(* Schneider Machine Expert - Basic project meccanismo_scelta_spegnimento_graduale_o_livello_minimo, file version 3.0.0.0 *)
(* ProjectInformations: Name=New project *)

HARDWARE
  Cpu 0: TM221C40R
  ModuleExtensionObject 0: TM3AI8/G
  EthernetConfiguration: NetworkName=M221, IpAllocationMode=FixedAddress, IpAddress=0.0.0.0, SubnetMask=0.0.0.0
  SerialLineConfiguration: Baud=Baud19200, Parity=ParityEven, DataBits=DataBits8, StopBits=StopBits1, PhysicalMedium=PhysicalMediumRs485, TransmissionMode=TransmissionModeModbusRtu, SlaveId=1, Addressing=SlaveAddressing
  MastTask: UsePeriodScanMode=false, PeriodScan=100
  FastTask: Period=255
  CpuBehavior: StartingMode=StartAsPreviousState, AutoSaveRamOnEeprom=true, WatchdogPeriod=250

SYMBOLS  (address, symbol, comment, settings)
  %M0       P1_USABILE
  %M1       P2_USABILE
  %M2       P1_COMANDATA  "Stesso valore di P1_CMD. Permette di identificare gli edges, visto che P1_CMD non può farlo."
  %M3       P2_COMANDATA  "Stesso valore di P2_CMD. Permette di identificare gli edges, visto che P2_CMD non può farlo."
  %M4       P3_USABILE
  %M5       P4_USABILE
  %M6       P3_COMANDATA
  %M7       P4_COMANDATA
  %M8       ESISTE_PROX_POMPA_CON_MINOR_ORE  "Nel loop, può non esistere una prossima pompa usabile e non comandata con il minor numero ore."
  %M9       ORA_E_00  "E' mezzanotte?"
  %M10      DECISO_ORDINE  "In intervallo in cui alternare le pompe per altern. giorn., è stata deciso quale sarà prossima pompa con minor ore?"
  %M11      PRIMA_POMPA_COMANDATA  "La prima pompa dell'ordine è stata effettivamente comandata quando serviva?"
  %M12      SECONDA_POMPA_COMANDATA  "La seconda pompa dell'ordine è stata effettivamente comandata quando serviva?"
  %M13      TERZA_POMPA_COMANDATA  "La terza pompa dell'ordine è stata effettivamente comandata quando serviva?"
  %M14      SOTTO_SOGLIA_MIN1
  %M15      SOPRA_SOGLIA_MAX1
  %M16      SOPRA_SOGLIA_MAX2
  %M17      PASSATO_SOGLIA_MAX1
  %M18      PASSATO_SOGLIA_MAX2
  %M19      SOTTO_SOGLIA_MIN2
  %M20      PASSATO_SOGLIA_MAX3
  %M21      PASSATO_SOGLIA_MIN3
  %M22      SOTTO_SOGLIA_MIN3
  %M23      SOPRA_SOGLIA_MAX3
  %M24      P5_USABILE
  %M25        "(occupato, placeholder)"
  %M26      P6_USABILE
  %M27      P5_COMANDATA
  %M28      P6_COMANDATA
  %M29      QUARTA_POMPA_COMANDATA
  %M30      QUINTA_POMPA_COMANDATA
  %M100       "(occupato, placeholder)"
  %MW0      NUM_POMPE_DA_COMANDARE  "Numero di pompe da comandare in base alle soglie raggiunte."
  %MW1      NUM_POMPE_COMANDATE  "Numero di pompe effettivamente comandate, in base alle loro disponibilità."
  %MW2      NUM_POMPE  "Numero di pompe totali."
  %MW3      ULTIMO_MINOR_SECONDI_LAVORATI  "Ultimi secondi lavorati più piccoli (valore temporaneo, da usare solo nel loop)."
  %MW4      PROSSIMA_POMPA_DA_COMANDARE  "Numero da 1 a NUM_POMPE che indica la prossima pompa da comandare."
  %MW5      POMPA_ATTUALE_LOOP  "Pompa attuale nel loop."
  %MW6      NUM_POMPE_COMANDATE_MAX  "Num"
  %MW7      CONTA_POMPE_COMANDATE_MAX  "Da usare in loop e da resettare.  Assume il valore da 1 fino a NUM_POMPE_COMANDATE_MAX."
  %MW8      ORDINE_PRIMA_POMPA
  %MW9      ORDINE_SECONDA_POMPA
  %MW10     ORDINE_TERZA_POMPA
  %MW11     STRG_ALTERNANZA_ATTUALE
  %MW12     LVL_PERC
  %MW13     ORDINE_QUARTA_POMPA
  %MW14     ORDINE_QUINTA_POMPA
  %C0       CONTATORE_P1_SECONDI_LAVORATI  [Preset=0]
  %C1       CONTATORE_P2_SECONDI_LAVORATI  [Preset=0]
  %C2       CONTATORE_P3_SECONDI_LAVORATI  [Preset=0]
  %C3       CONTATORE_P4_SECONDI_LAVORATI  [Preset=0]
  %C4       CONTATORE_P5_SECONDI_LAVORATI  [Preset=0]
  %C5       CONTATORE_P6_SECONDI_LAVORATI  [Preset=0]
  %I0.0     P1_AUTO
  %I0.1     P1_MOTO
  %I0.2     P1_ANOMALIA
  %I0.3     P2_AUTO
  %I0.4     P2_MOTO
  %I0.5     P2_ANOMALIA
  %I0.9     P3_AUTO
  %I0.10    P3_MOTO
  %I0.11    P3_ANOMALIA
  %I0.12    P4_AUTO
  %I0.13    P4_MOTO
  %I0.14    P4_ANOMALIA
  %I0.15    P5_AUTO
  %I0.16    P5_MOTO
  %I0.17    P5_ANOMALIA
  %I0.18    P6_AUTO
  %I0.19    P6_MOTO
  %I0.20    P6_ANOMALIA
  %Q0.0     P1_CMD
  %Q0.1     P2_CMD
  %Q0.2     P3_CMD
  %Q0.3     P4_CMD
  %Q0.4     ERR_STRG_ALTERNANZA_INVALIDA
  %Q0.5     P5_CMD
  %Q0.6     P6_CMD
  %IW0.0    IO_STRG_ALTERNANZA  "0 = livello minimo; 1 = spegnimento graduale;"  [Type=Type_0_10V, Scope=Scope_Normal, Minimum=0, Maximum=1000]
  %IW1.0    IO_LVL  [Type=Type_4_20mA, Scope=Scope_Customized, Minimum=4000, Maximum=20000]
  %IW1.1    SOGLIA_MIN1_PERC  [Type=Type_0_10V, Scope=Scope_Customized, Minimum=0, Maximum=100]
  %IW1.2    SOGLIA_MAX1_PERC  [Type=Type_0_10V, Scope=Scope_Customized, Minimum=0, Maximum=100]
  %IW1.3    SOGLIA_MIN2_PERC  [Type=Type_0_10V, Scope=Scope_Customized, Minimum=0, Maximum=100]
  %IW1.4    SOGLIA_MAX2_PERC  [Type=Type_0_10V, Scope=Scope_Customized, Minimum=0, Maximum=100]
  %IW1.5    SOGLIA_MIN3_PERC  [Type=Type_0_10V, Scope=Scope_Customized, Minimum=0, Maximum=100]
  %IW1.6    SOGLIA_MAX3_PERC  [Type=Type_0_10V, Scope=Scope_Customized, Minimum=0, Maximum=100]

POU Main
  (* SectionNumber=1 *)

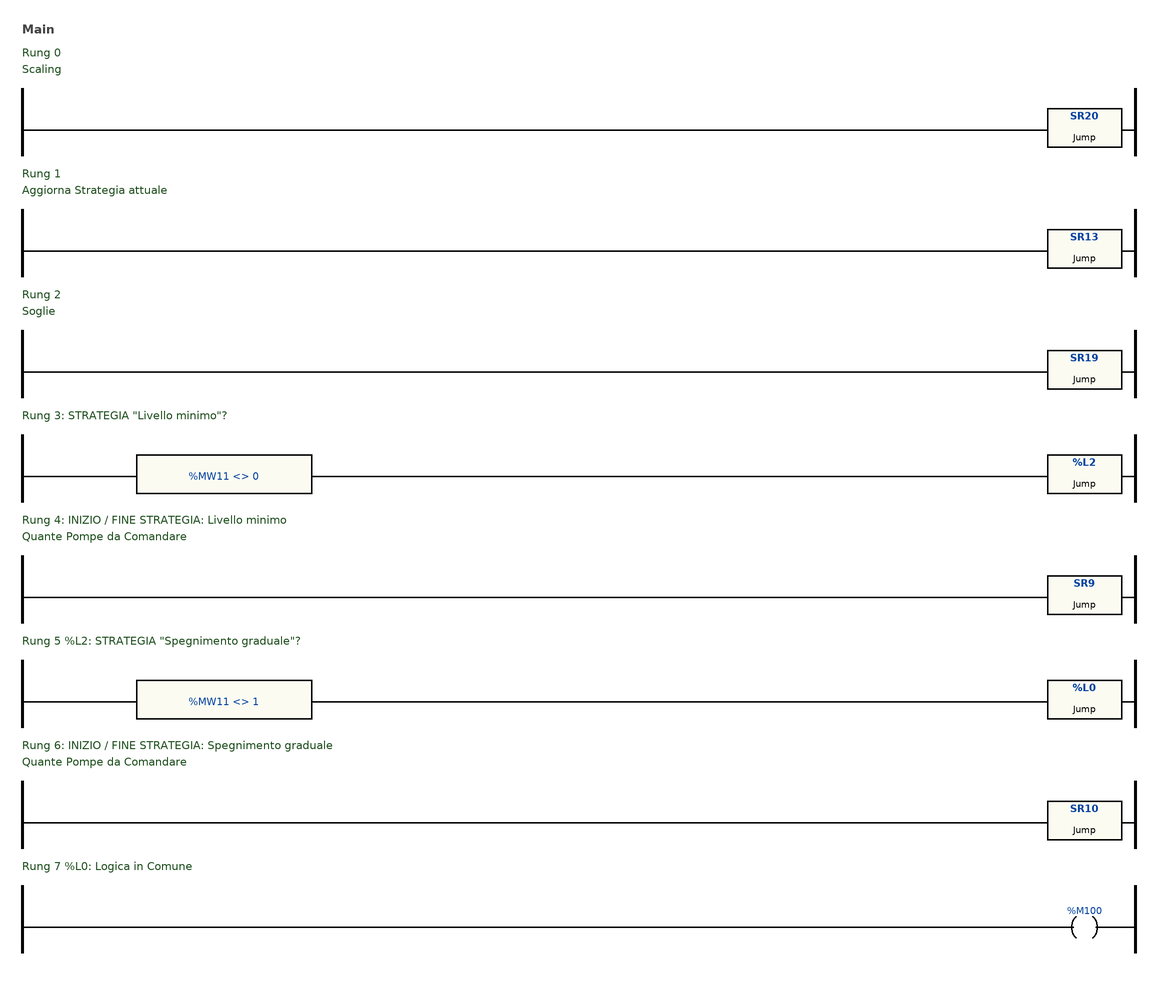

// Rung 0
// Scaling
  LD 1
  SR20
  // as ST:
  //   SR20();

// Rung 1
// Aggiorna Strategia attuale
  LD 1
  SR13
  // as ST:
  //   SR13();

// Rung 2
// Soglie
  LD 1
  SR19
  // as ST:
  //   SR19();

// Rung 3: STRATEGIA "Livello minimo"?
  LD [ %MW11 <> 0 ]       (* STRG_ALTERNANZA_ATTUALE *)
  JMPC %L2
  // as ST:
  //   IF STRG_ALTERNANZA_ATTUALE <> 0 THEN JMP %L2; END_IF;

// Rung 4: INIZIO / FINE STRATEGIA: Livello minimo
// Quante Pompe da Comandare
  LD 1
  SR9
  // as ST:
  //   SR9();

// Rung 5 %L2: STRATEGIA "Spegnimento graduale"?
  %L2:
  LD [ %MW11 <> 1 ]       (* STRG_ALTERNANZA_ATTUALE *)
  JMPC %L0
  // as ST:
  //   %L2:
  //   IF STRG_ALTERNANZA_ATTUALE <> 1 THEN JMP %L0; END_IF;

// Rung 6: INIZIO / FINE STRATEGIA: Spegnimento graduale
// Quante Pompe da Comandare
  LD 1
  SR10
  // as ST:
  //   SR10();

// Rung 7 %L0: Logica in Comune
  %L0:
  LD 1
  ST %M100
  // as ST:
  //   %L0:
  //   %M100 := TRUE;

Subroutine Aggiorna Strategia Alternanza
  (* SectionNumber=11, Number=13 *)

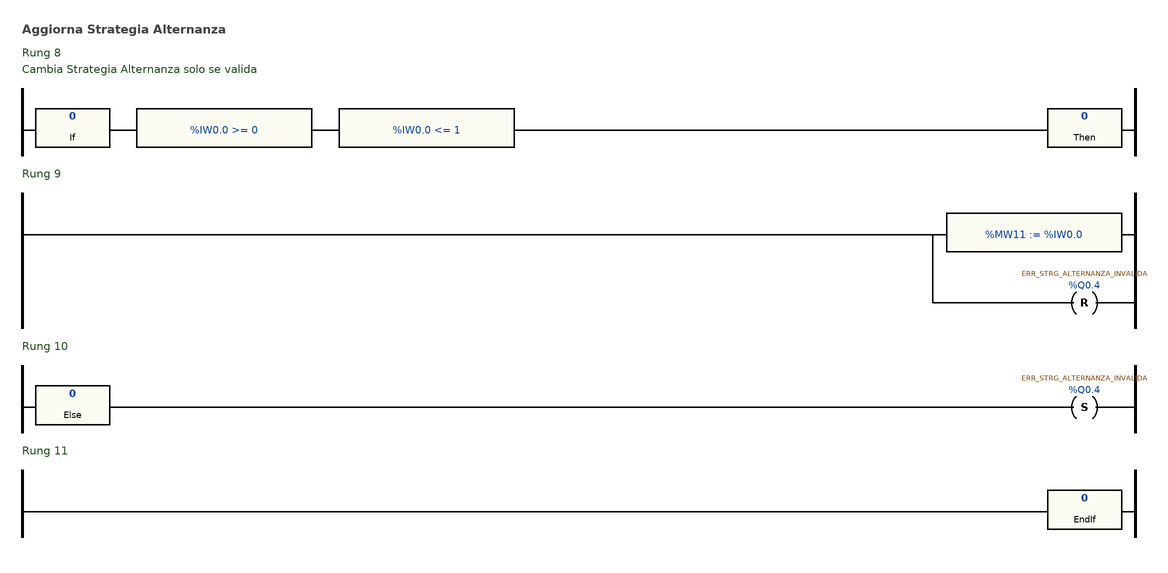

// Rung 8
// Cambia Strategia Alternanza solo se valida
  IF0
  AND [ %IW0.0 >= 0 ]     (* IO_STRG_ALTERNANZA *)
  AND [ %IW0.0 <= 1 ]     (* IO_STRG_ALTERNANZA *)
  THEN0

// Rung 9
  LD 1
  [ %MW11 := %IW0.0 ]     (* STRG_ALTERNANZA_ATTUALE, IO_STRG_ALTERNANZA *)
  R %Q0.4                 (* ERR_STRG_ALTERNANZA_INVALIDA *)
  // as ST:
  //   STRG_ALTERNANZA_ATTUALE := IO_STRG_ALTERNANZA;
  //   ERR_STRG_ALTERNANZA_INVALIDA := FALSE;

// Rung 10
  ELSE0
  S %Q0.4                 (* ERR_STRG_ALTERNANZA_INVALIDA *)

// Rung 11
  LD 1
  ENDIF0

Subroutine Soglie
  (* SectionNumber=12, Number=19 *)

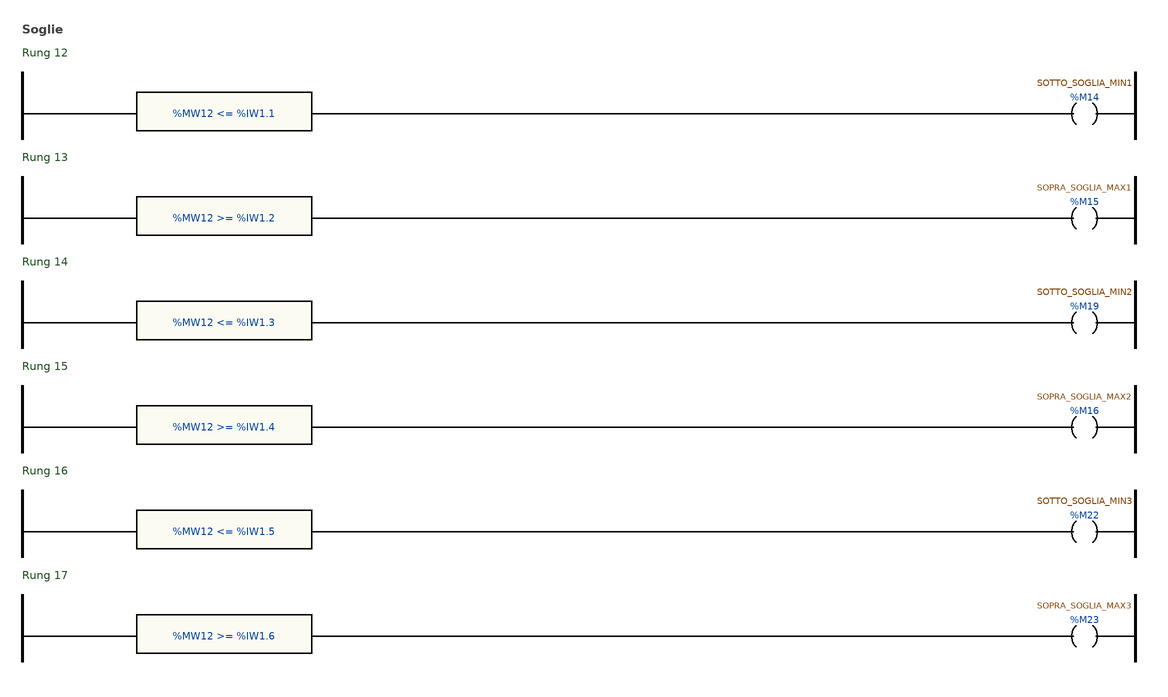

// Rung 12
  LD [ %MW12 <= %IW1.1 ]  (* LVL_PERC, SOGLIA_MIN1_PERC *)
  ST %M14                 (* SOTTO_SOGLIA_MIN1 *)
  // as ST:
  //   SOTTO_SOGLIA_MIN1 := LVL_PERC <= SOGLIA_MIN1_PERC;

// Rung 13
  LD [ %MW12 >= %IW1.2 ]  (* LVL_PERC, SOGLIA_MAX1_PERC *)
  ST %M15                 (* SOPRA_SOGLIA_MAX1 *)
  // as ST:
  //   SOPRA_SOGLIA_MAX1 := LVL_PERC >= SOGLIA_MAX1_PERC;

// Rung 14
  LD [ %MW12 <= %IW1.3 ]  (* LVL_PERC, SOGLIA_MIN2_PERC *)
  ST %M19                 (* SOTTO_SOGLIA_MIN2 *)
  // as ST:
  //   SOTTO_SOGLIA_MIN2 := LVL_PERC <= SOGLIA_MIN2_PERC;

// Rung 15
  LD [ %MW12 >= %IW1.4 ]  (* LVL_PERC, SOGLIA_MAX2_PERC *)
  ST %M16                 (* SOPRA_SOGLIA_MAX2 *)
  // as ST:
  //   SOPRA_SOGLIA_MAX2 := LVL_PERC >= SOGLIA_MAX2_PERC;

// Rung 16
  LD [ %MW12 <= %IW1.5 ]  (* LVL_PERC, SOGLIA_MIN3_PERC *)
  ST %M22                 (* SOTTO_SOGLIA_MIN3 *)
  // as ST:
  //   SOTTO_SOGLIA_MIN3 := LVL_PERC <= SOGLIA_MIN3_PERC;

// Rung 17
  LD [ %MW12 >= %IW1.6 ]  (* LVL_PERC, SOGLIA_MAX3_PERC *)
  ST %M23                 (* SOPRA_SOGLIA_MAX3 *)
  // as ST:
  //   SOPRA_SOGLIA_MAX3 := LVL_PERC >= SOGLIA_MAX3_PERC;

Subroutine Scaling
  (* SectionNumber=13, Number=20 *)

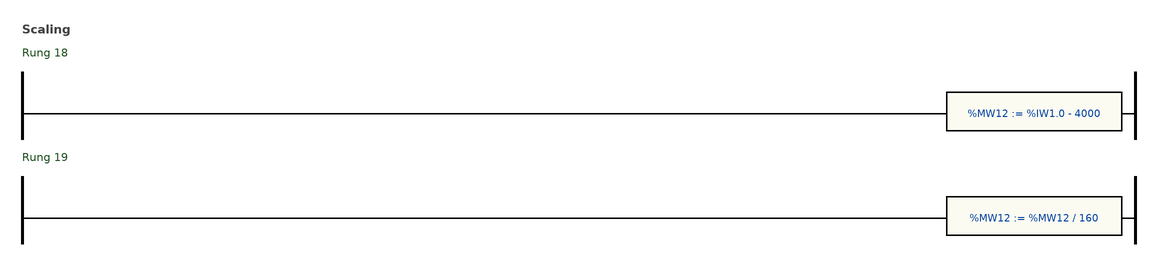

// Rung 18
  LD 1
  [ %MW12 := %IW1.0 - 4000 ](* LVL_PERC, IO_LVL *)
  // as ST:
  //   LVL_PERC := IO_LVL - 4000;

// Rung 19
  LD 1
  [ %MW12 := %MW12 / 160 ](* LVL_PERC, LVL_PERC *)
  // as ST:
  //   LVL_PERC := LVL_PERC / 160;

Subroutine Quante Pompe da Comandare (Livello minimo)
  (* SectionNumber=14, Number=9 *)

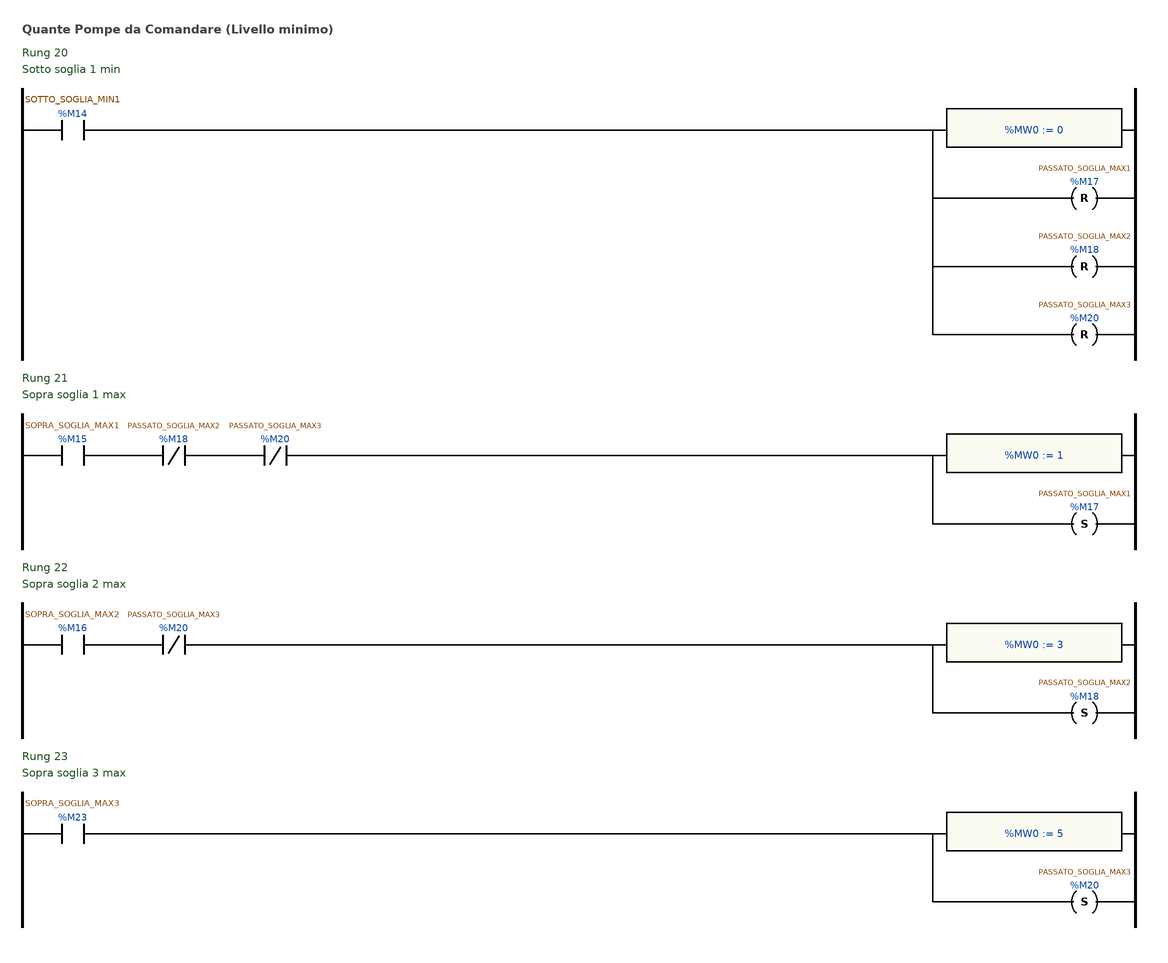

// Rung 20
// Sotto soglia 1 min
  LD %M14                 (* SOTTO_SOGLIA_MIN1 *)
  [ %MW0 := 0 ]           (* NUM_POMPE_DA_COMANDARE *)
  R %M17                  (* PASSATO_SOGLIA_MAX1 *)
  R %M18                  (* PASSATO_SOGLIA_MAX2 *)
  R %M20                  (* PASSATO_SOGLIA_MAX3 *)
  // as ST:
  //   IF SOTTO_SOGLIA_MIN1 THEN NUM_POMPE_DA_COMANDARE := 0; END_IF;
  //   IF SOTTO_SOGLIA_MIN1 THEN PASSATO_SOGLIA_MAX1 := FALSE; END_IF;
  //   IF SOTTO_SOGLIA_MIN1 THEN PASSATO_SOGLIA_MAX2 := FALSE; END_IF;
  //   IF SOTTO_SOGLIA_MIN1 THEN PASSATO_SOGLIA_MAX3 := FALSE; END_IF;

// Rung 21
// Sopra soglia 1 max
  LD %M15                 (* SOPRA_SOGLIA_MAX1 *)
  ANDN %M18               (* PASSATO_SOGLIA_MAX2 *)
  ANDN %M20               (* PASSATO_SOGLIA_MAX3 *)
  [ %MW0 := 1 ]           (* NUM_POMPE_DA_COMANDARE *)
  S %M17                  (* PASSATO_SOGLIA_MAX1 *)
  // as ST:
  //   IF SOPRA_SOGLIA_MAX1 AND NOT PASSATO_SOGLIA_MAX2 AND NOT PASSATO_SOGLIA_MAX3 THEN NUM_POMPE_DA_COMANDARE := 1; END_IF;
  //   IF SOPRA_SOGLIA_MAX1 AND NOT PASSATO_SOGLIA_MAX2 AND NOT PASSATO_SOGLIA_MAX3 THEN PASSATO_SOGLIA_MAX1 := TRUE; END_IF;

// Rung 22
// Sopra soglia 2 max
  LD %M16                 (* SOPRA_SOGLIA_MAX2 *)
  ANDN %M20               (* PASSATO_SOGLIA_MAX3 *)
  [ %MW0 := 3 ]           (* NUM_POMPE_DA_COMANDARE *)
  S %M18                  (* PASSATO_SOGLIA_MAX2 *)
  // as ST:
  //   IF SOPRA_SOGLIA_MAX2 AND NOT PASSATO_SOGLIA_MAX3 THEN NUM_POMPE_DA_COMANDARE := 3; END_IF;
  //   IF SOPRA_SOGLIA_MAX2 AND NOT PASSATO_SOGLIA_MAX3 THEN PASSATO_SOGLIA_MAX2 := TRUE; END_IF;

// Rung 23
// Sopra soglia 3 max
  LD %M23                 (* SOPRA_SOGLIA_MAX3 *)
  [ %MW0 := 5 ]           (* NUM_POMPE_DA_COMANDARE *)
  S %M20                  (* PASSATO_SOGLIA_MAX3 *)
  // as ST:
  //   IF SOPRA_SOGLIA_MAX3 THEN NUM_POMPE_DA_COMANDARE := 5; END_IF;
  //   IF SOPRA_SOGLIA_MAX3 THEN PASSATO_SOGLIA_MAX3 := TRUE; END_IF;

Subroutine Quante Pompe da Comandare (Spegnimento graduale)
  (* SectionNumber=15, Number=10 *)

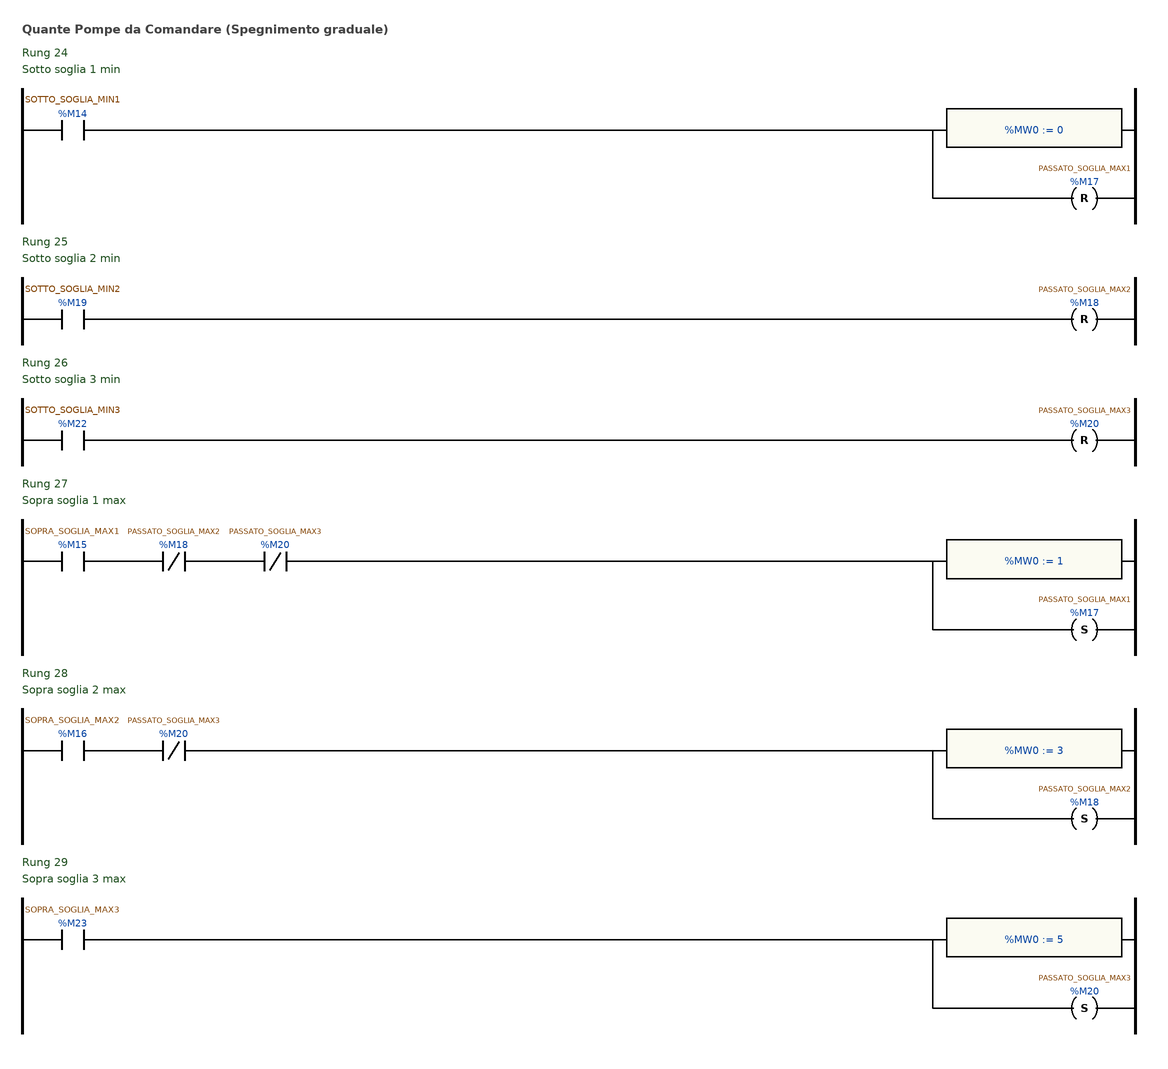

// Rung 24
// Sotto soglia 1 min
  LD %M14                 (* SOTTO_SOGLIA_MIN1 *)
  [ %MW0 := 0 ]           (* NUM_POMPE_DA_COMANDARE *)
  R %M17                  (* PASSATO_SOGLIA_MAX1 *)
  // as ST:
  //   IF SOTTO_SOGLIA_MIN1 THEN NUM_POMPE_DA_COMANDARE := 0; END_IF;
  //   IF SOTTO_SOGLIA_MIN1 THEN PASSATO_SOGLIA_MAX1 := FALSE; END_IF;

// Rung 25
// Sotto soglia 2 min
  LD %M19                 (* SOTTO_SOGLIA_MIN2 *)
  R %M18                  (* PASSATO_SOGLIA_MAX2 *)
  // as ST:
  //   IF SOTTO_SOGLIA_MIN2 THEN PASSATO_SOGLIA_MAX2 := FALSE; END_IF;

// Rung 26
// Sotto soglia 3 min
  LD %M22                 (* SOTTO_SOGLIA_MIN3 *)
  R %M20                  (* PASSATO_SOGLIA_MAX3 *)
  // as ST:
  //   IF SOTTO_SOGLIA_MIN3 THEN PASSATO_SOGLIA_MAX3 := FALSE; END_IF;

// Rung 27
// Sopra soglia 1 max
  LD %M15                 (* SOPRA_SOGLIA_MAX1 *)
  ANDN %M18               (* PASSATO_SOGLIA_MAX2 *)
  ANDN %M20               (* PASSATO_SOGLIA_MAX3 *)
  [ %MW0 := 1 ]           (* NUM_POMPE_DA_COMANDARE *)
  S %M17                  (* PASSATO_SOGLIA_MAX1 *)
  // as ST:
  //   IF SOPRA_SOGLIA_MAX1 AND NOT PASSATO_SOGLIA_MAX2 AND NOT PASSATO_SOGLIA_MAX3 THEN NUM_POMPE_DA_COMANDARE := 1; END_IF;
  //   IF SOPRA_SOGLIA_MAX1 AND NOT PASSATO_SOGLIA_MAX2 AND NOT PASSATO_SOGLIA_MAX3 THEN PASSATO_SOGLIA_MAX1 := TRUE; END_IF;

// Rung 28
// Sopra soglia 2 max
  LD %M16                 (* SOPRA_SOGLIA_MAX2 *)
  ANDN %M20               (* PASSATO_SOGLIA_MAX3 *)
  [ %MW0 := 3 ]           (* NUM_POMPE_DA_COMANDARE *)
  S %M18                  (* PASSATO_SOGLIA_MAX2 *)
  // as ST:
  //   IF SOPRA_SOGLIA_MAX2 AND NOT PASSATO_SOGLIA_MAX3 THEN NUM_POMPE_DA_COMANDARE := 3; END_IF;
  //   IF SOPRA_SOGLIA_MAX2 AND NOT PASSATO_SOGLIA_MAX3 THEN PASSATO_SOGLIA_MAX2 := TRUE; END_IF;

// Rung 29
// Sopra soglia 3 max
  LD %M23                 (* SOPRA_SOGLIA_MAX3 *)
  [ %MW0 := 5 ]           (* NUM_POMPE_DA_COMANDARE *)
  S %M20                  (* PASSATO_SOGLIA_MAX3 *)
  // as ST:
  //   IF SOPRA_SOGLIA_MAX3 THEN NUM_POMPE_DA_COMANDARE := 5; END_IF;
  //   IF SOPRA_SOGLIA_MAX3 THEN PASSATO_SOGLIA_MAX3 := TRUE; END_IF;
